// TIA Portal V21 export
FUNCTION "deviceState" : Void   // FC904, LAD
{ S7_Optimized_Access := 'TRUE' }
// stored: AutoNumber false, SetENOAutomatically false
   VAR_INPUT
      Alarm : Bool;
      Warning : Bool;
      Running : Bool;
      Reverse : Bool;
      Service : Bool;
   END_VAR
   VAR_IN_OUT
      deviceIcon : Int;
   END_VAR
BEGIN

REGION Network 1
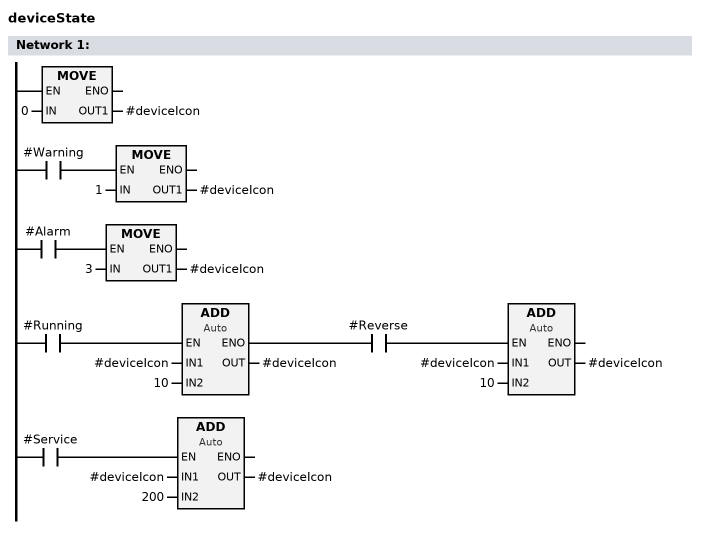
   RUNG wire#powerrail
      Move(in := 0, out1 => #deviceIcon)
   END_RUNG
   RUNG wire#powerrail
      Contact( #Warning )
      Move(in := 1, out1 => #deviceIcon)
   END_RUNG
   RUNG wire#powerrail
      Contact( #Alarm )
      Move(in := 3, out1 => #deviceIcon)
   END_RUNG
   RUNG wire#powerrail
      Contact( #Running )
      Add(in1 := #deviceIcon, in2 := 10, out => #deviceIcon)
      Contact( #Reverse )
      Add(in1 := #deviceIcon, in2 := 10, out => #deviceIcon)
   END_RUNG
   RUNG wire#powerrail
      Contact( #Service )
      Add(in1 := #deviceIcon, in2 := 200, out => #deviceIcon)
   END_RUNG
   // the same network as SCL:
   #deviceIcon := 0;
   IF #Warning THEN #deviceIcon := 1; END_IF;
   IF #Alarm THEN #deviceIcon := 3; END_IF;
   IF #Running THEN #deviceIcon := #deviceIcon + 10; END_IF;
   IF #Running AND #Reverse THEN #deviceIcon := #deviceIcon + 10; END_IF;
   IF #Service THEN #deviceIcon := #deviceIcon + 200; END_IF;
END_REGION
END_FUNCTION
